// TIA Portal V19 export
DATA_BLOCK "DriveLogic_DB"   // DB4
// stored: InstanceOfName DriveLogic, InstanceOfType FB
"DriveLogic"
   // VAR_INPUT
   //    Enable_Drives : Bool;
   //    AckError : Bool;
   //    SpeedSp : Real;
   // END_VAR
   // VAR
   //    SINA_SPEED_Instance_1 : "SINA_SPEED";
   // END_VAR
BEGIN
END_DATA_BLOCK
